(* CoDeSys 2.3.5.6 project: szlendak_01.pro *)
(* Libraries: Standard.lib*4.1.15 16:23:13, SYSLIBCALLBACK.LIB*4.1.15 16:23:13 *)

(* PLC configuration (modules and I/O channels)
I1 AT %IX0.0 [LocalBitInput] Input I1
I2 AT %IX0.1 [LocalBitInput] Input I2
I3 AT %IX0.2 [LocalBitInput] Input I3
I4 AT %IX0.3 [LocalBitInput] Input I4
I5 AT %IX0.4 [LocalBitInput] Input I5
I6 AT %IX0.5 [LocalBitInput] Input I6
I7 AT %IX0.6 [LocalBitInput] Input I7
I8 AT %IX0.7 [LocalBitInput] Input I8
I9 AT %IX1.0 [LocalBitInput] Input I9
I10 AT %IX1.1 [LocalBitInput] Input I10
I11 AT %IX1.2 [LocalBitInput] Input I11
I12 AT %IX1.3 [LocalBitInput] Input I12
I13 AT %IX1.4 [LocalDiagInput] Diagnostic Input I13
I14 AT %IX1.5 [LocalDiagInput] Diagnostic Input I14
I15 AT %IX1.6 [LocalDiagInput] Diagnostic Input I15
I16 AT %IX1.7 [LocalDiagInput] Diagnostic Input I16
I7_Analog AT %IW2 [LocalAnalogIn] Input I7, 10Bit, 0-10VDC
I8_Analog AT %IW4 [LocalAnalogIn] Input I8, 10Bit, 0-10VDC
I11_Analog AT %IW6 [LocalAnalogIn] Input I11, 10Bit, 0-10VDC
I12_Analog AT %IW8 [LocalAnalogIn] Input I12, 10Bit, 0-10VDC
Q1 AT %QX0.0 [LocalBitOutput] Transistor-Output Q1
Q2 AT %QX0.1 [LocalBitOutput] Transistor-Output Q2
Q3 AT %QX0.2 [LocalBitOutput] Transistor-Output Q3
Q4 AT %QX0.3 [LocalBitOutput] Transistor-Output Q4
Q5 AT %QX0.4 [LocalBitOutput] Transistor-Output Q5
Q6 AT %QX0.5 [LocalBitOutput] Transistor-Output Q6
Q7 AT %QX0.6 [LocalBitOutput] Transistor-Output Q7
Q8 AT %QX0.7 [LocalBitOutput] Transistor-Output Q8
No Analog Output [EC4P_NoAnalogOutput] node 1, in %IB10 out %QB1
No Keys [EC4P_NoKeys] node 2, in %IB10 out %QB1
No Counter [EC4P_NoCounter] node 3, in %IB10 out %QB1
Extension [EC4P_Extension] node 1, in %IB10 out %QB1
  No Extension [EC4P_NoExtension] node 0, in %IB10 out %QB1
*)

(* POU PLC_PRG, LD *)
PROGRAM PLC_PRG
VAR
END_VAR
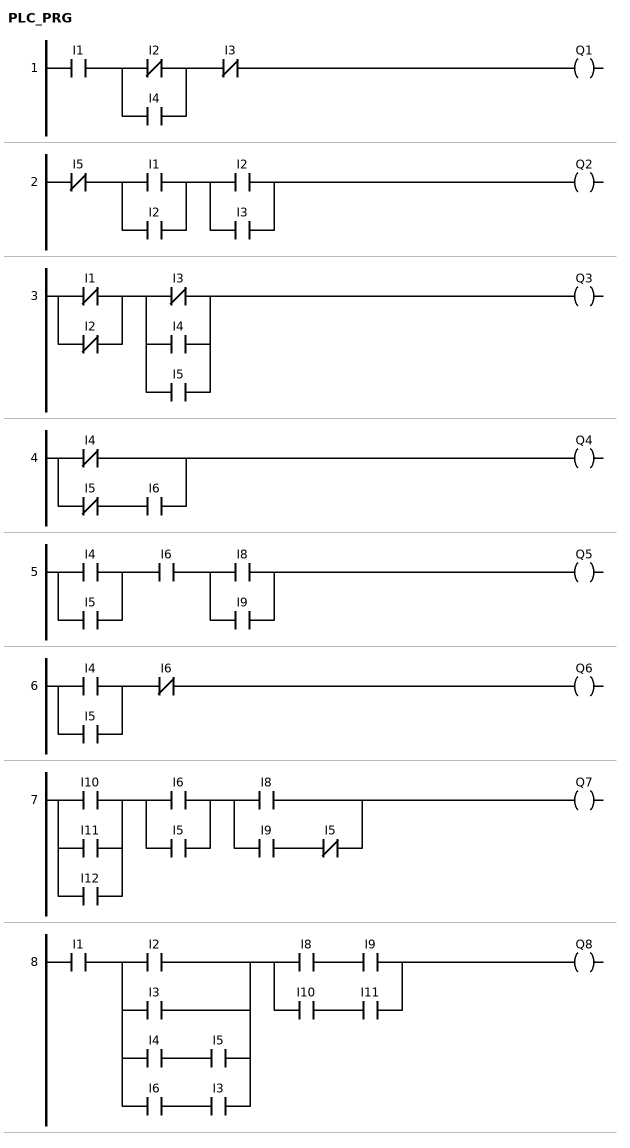
_LD_ (* Ladder Diagram *)
NETWORK 1
	[I1] - { [/I2] | [I4] } - [/I3] --- (Q1)
NETWORK 2
	[/I5] - { [I1] | [I2] } - { [I2] | [I3] } --- (Q2)
NETWORK 3
	{ [/I1] | [/I2] } - { [/I3] | [I4] | [I5] } --- (Q3)
NETWORK 4
	{ [/I4] | [/I5] - [I6] } --- (Q4)
NETWORK 5
	{ [I4] | [I5] } - [I6] - { [I8] | [I9] } --- (Q5)
NETWORK 6
	{ [I4] | [I5] } - [/I6] --- (Q6)
NETWORK 7
	{ [I10] | [I11] | [I12] } - { [I6] | [I5] } - { [I8] | [I9] - [/I5] } --- (Q7)
NETWORK 8
	[I1] - { [I2] | [I3] | [I4] - [I5] | [I6] - [I3] } - { [I8] - [I9] | [I10] - [I11] } --- (Q8)
_END_LD_
(* the same logic as Structured Text *)
(* Network 1 *)
Q1 := I1 AND (NOT I2 OR I4) AND NOT I3;
(* Network 2 *)
Q2 := NOT I5 AND (I1 OR I2) AND (I2 OR I3);
(* Network 3 *)
Q3 := (NOT I1 OR NOT I2) AND (NOT I3 OR I4 OR I5);
(* Network 4 *)
Q4 := NOT I4 OR NOT I5 AND I6;
(* Network 5 *)
Q5 := (I4 OR I5) AND I6 AND (I8 OR I9);
(* Network 6 *)
Q6 := (I4 OR I5) AND NOT I6;
(* Network 7 *)
Q7 := (I10 OR I11 OR I12) AND (I6 OR I5) AND (I8 OR I9 AND NOT I5);
(* Network 8 *)
Q8 := I1 AND (I2 OR I3 OR I4 AND I5 OR I6 AND I3) AND (I8 AND I9 OR I10 AND I11);
END_PROGRAM
